PROGRAM MAIN
VAR
	fbValve		:	FB_ControlValve;
	CurrentDat	:	ST_ValveDat;
END_VAR

TestModbus();
fbValve(fSetPerc:=5000,fAct=>CurrentDat); //50.00%

END_PROGRAM

(* stored: Version 1.1.0.1, ProductVersion 3.1.4022.10
   POU MAIN: Id {602de947-c890-43bc-9e37-71712f8ad59a}, SpecialFunc None *)
